FUNCTION_BLOCK FB_RV_Output
VAR_INPUT
	Betrieb				:BOOL;
	Stellung			:USINT;
END_VAR
VAR_OUTPUT
	OUT_Stellung		: INT;
END_VAR
VAR
END_VAR

OUT_Stellung 		:= USINT_TO_INT(Stellung) * 327;

END_FUNCTION_BLOCK

(* stored: Version 1.1.0.1, ProductVersion 3.1.4024.9
   POU FB_RV_Output: Id {e967feef-cb0c-42fd-a763-38ed25b3797d}, SpecialFunc None *)
